// TIA Portal V18 export
FUNCTION_BLOCK "Main_Safety_RTG1"   // FB1, F_FBD
{ S7_Optimized_Access := 'TRUE' }
// stored: AutoNumber false
   VAR_TEMP
      t_Reset : Bool;
   END_VAR
   VAR_TEMP   // added for the SCL form of the ladder/FBD networks
      _w1 : Bool;
      _w2 : Bool;
   END_VAR
BEGIN

REGION Network 1: For commissioning
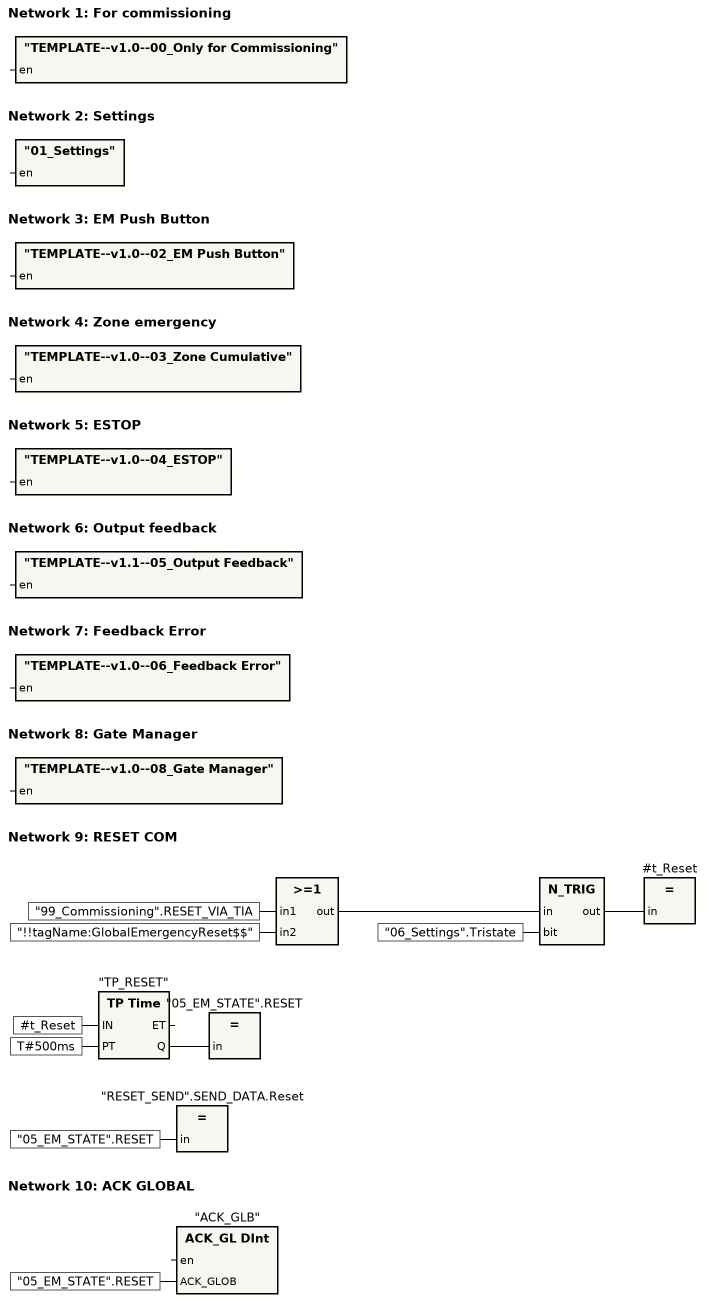
   "TEMPLATE--v1.0--00_Only for Commissioning"();
END_REGION

REGION Network 2: Settings
   "01_Settings"();
END_REGION

REGION Network 3: EM Push Button
   "TEMPLATE--v1.0--02_EM Push Button"();
END_REGION

REGION Network 4: Zone emergency
   "TEMPLATE--v1.0--03_Zone Cumulative"();
END_REGION

REGION Network 5: ESTOP
   "TEMPLATE--v1.0--04_ESTOP"();
END_REGION

REGION Network 6: Output feedback
   "TEMPLATE--v1.1--05_Output Feedback"();
END_REGION

REGION Network 7: Feedback Error
   "TEMPLATE--v1.0--06_Feedback Error"();
END_REGION

REGION Network 8: Gate Manager
   "TEMPLATE--v1.0--08_Gate Manager"();
END_REGION

REGION Network 9: RESET COM
   // Add any other reset
   #_w1 := "99_Commissioning".RESET_VIA_TIA OR "!!tagName:GlobalEmergencyReset$$";
   #_w2 := NOT #_w1 AND "06_Settings".Tristate;   // falling edge
   "06_Settings".Tristate := #_w1;
   #t_Reset := #_w2;
   "TP_RESET".TP(IN := #t_Reset, PT := T#500ms);
   "05_EM_STATE".RESET := "TP_RESET".Q;
   "RESET_SEND".SEND_DATA.Reset := "05_EM_STATE".RESET;
END_REGION

REGION Network 10: ACK GLOBAL
   "ACK_GLB"(ACK_GLOB := "05_EM_STATE".RESET);   // ACK_GL
END_REGION
END_FUNCTION_BLOCK
